FUNCTION_BLOCK NotifierEvent EXTENDS R_TRIG
VAR_INPUT
	sModuleName : T_MaxString;
	sDeviceName : T_MaxString;
	sStatus: T_MaxString;
	sMessage : T_MaxString;
END_VAR
VAR_IN_OUT
	fbNotifier : Notifier;
END_VAR
VAR_OUTPUT
END_VAR
VAR
	
END_VAR

SUPER^();
IF 		Q
	AND __ISVALIDREF(fbNotifier)
THEN
	fbNotifier.Write(
		sDeviceName := sDeviceName,
		sMessage := sMessage,
		sModuleName := sModuleName,
		sStatus := sStatus);
END_IF

END_FUNCTION_BLOCK

(* stored: Version 1.1.0.1, ProductVersion 3.1.4024.2
   POU NotifierEvent: Id {e22bd0c9-9993-4c66-9376-3ddb1028b9e6}, SpecialFunc None *)
